% RSLogix 500 project Tarea_5_semaforo_secuenciador_PLC.RSS, saved by version 8.30.00.16 %
PROJECT "UNTITLED"    % processor: MicroLogix 1000 %

PROGRAM FILES
  LAD 2 "MAIN_PROG"  4 rungs
  LAD 3 "USER_FAULT"  1 rungs
  LAD 4 "HSC_INT"  1 rungs
  LAD 5 "STI_INT"  1 rungs
  LAD 6, 7, 8, 9, 10, 11, 12, 13, 14, 15, 16: only END

DATA FILES
  O0 OUTPUT  1 elements
  I1 INPUT  2 elements
  S2 STATUS  33 elements
  B3 BINARY  32 elements
  T4 TIMER  40 elements
  C5 COUNTER  32 elements
  R6 CONTROL  16 elements
  N7 INTEGER  105 elements

LADDER 2 "MAIN_PROG"
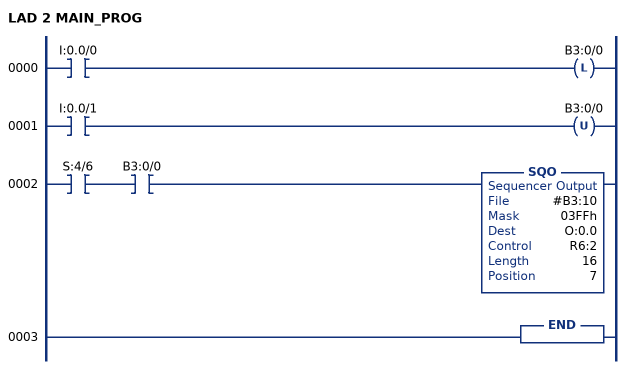
% Rung: 0 %
SOR XIC I:0.0/0 OTL B3:0/0 EOR
% Rung: 1 %
SOR XIC I:0.0/1 OTU B3:0/0 EOR
% Rung: 2 %
SOR XIC S:4/6 XIC B3:0/0 SQO #B3:10 03FFh O:0.0 R6:2 16 7 EOR
% Rung: 3 %
SOR END EOR

OTHER DOCUMENTED ADDRESSES
  B3:10/0  "0"

REVISION NOTES
  0: ya con registros

DATA TABLE (non-zero values as saved)
DATA B3
% B3:0 % 0X0001 0X0000 0X0000 0X0000 0X0000 0X0000 0X0000 0X0000 0X0000 0X0000
% B3:10 % 0X0000 0X0041 0X0041 0X0001 0X0041 0X0001 0X0041 0X0021 0X0021 0X0014
% B3:20 % 0X0014 0X0010 0X0014 0X0010 0X0014 0X0012 0X0012 0X0000 0X0000 0X0000
DATA R6
% .LEN .POS %
% R6:2 % 16 7
